ORGANIZATION_BLOCK MAIN:OB1
TITLE=PROGRAM COMMENTS
BEGIN
Network 1
LD     I0.1
LD     I2.0
O      I1.5
CTU    C1, 3
Network 2 //   Sıralı Çalıştırma
//   Tüm Devreyi Stoplama
LD     I1.5
O      I2.0
R      Q0.5, 10
R      T37, 2
R      M0.0, 3
Network 3
//   Start Verme
LDN    I0.0
A      C1
LD     I0.1
O      M0.0
ALD
=      M0.0
S      Q0.5, 1
R      Q1.2, 1
Network 4
//   İlk Döngü
LD     M0.0
A      Q0.5
TON    T37, 30
Network 5
//   İlk Döngü Sonucu
LD     T37
O      M0.1
R      Q0.5, 1


S      Q1.2, 1
S      M0.1, 1
R      T37, 1
R      M0.2, 1
Network 6
//   2. Döngü
LD     M0.0
A      Q1.2
TON    T38, 30
Network 7
//   2. Döngü Sonucu
LD     T38
O      M0.2
R      Q1.2, 1


S      Q0.5, 1
S      M0.2, 1
R      T38, 1
R      M0.1, 1
END_ORGANIZATION_BLOCK
SUBROUTINE_BLOCK SBR_0:SBR0
TITLE=SUBROUTINE COMMENTS
BEGIN
Network 1 //   Network Title
//   Network Comment
END_SUBROUTINE_BLOCK
INTERRUPT_BLOCK INT_0:INT0
TITLE=INTERRUPT ROUTINE COMMENTS
BEGIN
Network 1 //   Network Title
//   Network Comment
END_INTERRUPT_BLOCK
